PROGRAM MAIN
VAR
	//Config : ST_Configuration;
	VariantControl : FB_VariantControl;
	
	Cell : FB_Cell;
    HMI : FB_HMI;
END_VAR

// load machine config data
VariantControl(bLoadJSONFirstScan:=_TaskInfo[1].FirstCycle,
               bWriteJSON := HMI.HMItoPLC.variantControl.bExportJSON,
               Config := HMI.HMItoPLC.variantControl.Config);

// Don't execute anything until configuration data is loaded
IF VariantControl.bDone AND NOT VariantControl.bBusy THEN
    //Config := HMI.HMItoPLC.variantControl.Config;
    Cell(Config := HMI.HMItoPLC.variantControl.Config,
        HMItoPLC := HMI.HMItoPLC,
        PLCtoHMI => HMI.PLCtoHMI);

END_IF

// Run HMI as soon as machine config is loaded or failed to create config file
IF VariantControl.bDone THEN

    HMI.PLCtoHMI.variantControl.bNeedsCellDefinition := VariantControl.bLoadError;
    HMI();

END_IF

END_PROGRAM

(* stored: Version 1.1.0.1, ProductVersion 3.1.4024.9
   POU MAIN: Id {61fb59f7-cccf-4dc1-ac71-909a05e4fc8f}, SpecialFunc None *)
